TYPE E_MatchedMasterArmIdx :
(
	MatchedMasterArmIdx_NULL := 0,
	MatchedMasterArmIdx_Left := 1,
	MatchedMasterArmIdx_Right := 2
);
END_TYPE

(* stored: Version 1.1.0.1, ProductVersion 3.1.4024.12
   DUT E_MatchedMasterArmIdx: Id {7abc273c-3277-4ced-b2c2-72cdad391434} *)
